FUNCTION_BLOCK TcoInsight_v_5_x_x  EXTENDS TcoIo.TcoPnIoComponent 
VAR_IN_OUT
	inoIoData : TcoInsightIO_v_5_x_x;
END_VAR

VAR
	{attribute addProperty Name "<#Config#>"}
    _config : TcoInsightConfig_v_5_x_x;
	{attribute addProperty Name "<#Status#>"}
	_status : TcoInsightStatus_v_5_x_x;	
END_VAR

VAR
	{attribute addProperty Name "<#UserData#>"}
	_userData 	: TcoInsightUser_v_5_x_x;
	{attribute addProperty Name "<#Results#>"}
	_results : TcoInsightResults_v_5_x_x;
END_VAR

VAR
	{attribute 'hide'}
    _taskEnabled : BOOL;
	{attribute addProperty Name "<#Restore#>"}
    _restoreTask : TcoCore.TcoTask(THIS^);
	{attribute addProperty Name "<#Update signal states#>"}
    _updateSignalStatesTask : TcoCore.TcoTask(THIS^);
	{attribute addProperty Name "<#Change job by number#>"}
    _changeJobByNumberTask : TcoInsightChangeJobByNumber_v_5_x_x(THIS^);
	{attribute addProperty Name "<#Change job by name#>"}
    _changeJobByNameTask : TcoInsightChangeJobByName_v_5_x_x(THIS^);
	{attribute addProperty Name "<#Clear inspection results#>"}
    _clearInspectionResultsTask : TcoInsightClearInspectionResults_v_5_x_x(THIS^);
	{attribute addProperty Name "<#Set user data#>"}
    _setUserDataTask : TcoInsightSetUserData_v_5_x_x(THIS^);
	{attribute addProperty Name "<#Clear user data#>"}
    _clearUserDataTask : TcoInsightClearUserData_v_5_x_x(THIS^);
	{attribute addProperty Name "<#Soft event#>"}
    _softEventTask : TcoInsightSoftEvent_v_5_x_x(THIS^);
	{attribute addProperty Name "<#Trigger#>"}
    _triggerTask : TcoInsightTrigger_v_5_x_x(THIS^);
END_VAR
VAR
    {attribute 'hide'} 
	_varInfo : __SYSTEM.VAR_INFO;
    {attribute 'hide'} 
	_sb : TcoCore.StringBuilder;
END_VAR

IF InvalidReference() THEN
    RETURN;
END_IF

SUPER^(inPnIoBoxState := THIS^.inoIoData.PnIoBoxState,inPnIoBoxDiag := THIS^.inoIoData.PnIoBoxDiag);

IF NOT SUPER^.ProfinetReady THEN
	THIS^._status.ActionDescription := '<#Not ready for operation by means of Profinet network!#>';	
END_IF

IF SUPER^.ProfinetReady AND THIS^._status.ActionDescription = '<#Not ready for operation by means of Profinet network!#>' THEN
	THIS^._status.ActionDescription := '<#Ready for operation!#>';	
END_IF

CheckIfOnline();

//*************RESTORE********************
_taskEnabled := TRUE;
_restoreTask.Enabled := _taskEnabled;
IF _restoreTask.Execute() THEN
	Restore();
//	UpdateSignalStates();
END_IF
//****************************************

//*************UPDATE*********************
IF _config.UpdateStatesPermanently THEN
	UpdateSignalStates();
END_IF;

_taskEnabled:=SUPER^.ProfinetReady;
_taskEnabled := _taskEnabled AND NOT _restoreTask.Busy ;
_updateSignalStatesTask.Enabled := _taskEnabled;
IF _updateSignalStatesTask.Execute() THEN
	UpdateSignalStates();
END_IF
//****************************************

//*************CHANGE*JOB*BY*NUMBER*******
_taskEnabled:=SUPER^.ProfinetReady;
_taskEnabled := _taskEnabled AND NOT _updateSignalStatesTask.Busy;
_changeJobByNumberTask.Enabled := _taskEnabled;
_changeJobByNumberTask(inoIoData := THIS^.inoIoData,inoConfig := THIS^._config,inoStatus := THIS^._status);
//****************************************

//*************CHANGE*JOB*BY*NAME*********
_taskEnabled:=SUPER^.ProfinetReady;
_taskEnabled := _taskEnabled AND NOT _changeJobByNumberTask.Busy;
_changeJobByNameTask.Enabled := _taskEnabled;
_changeJobByNameTask(inoIoData := THIS^.inoIoData,inoConfig := THIS^._config,inoStatus := THIS^._status);
//****************************************

//*************CLEAR*DATA*****************
_taskEnabled:=SUPER^.ProfinetReady;
_taskEnabled := _taskEnabled AND NOT _changeJobByNameTask.Busy;
_clearInspectionResultsTask.Enabled := _taskEnabled;
_clearInspectionResultsTask(inoIoData := THIS^.inoIoData,inoConfig := THIS^._config,inoStatus := THIS^._status,inoResults := THIS^._results);
//****************************************

//*************CLEAR USER DATA*****************
_taskEnabled:=SUPER^.ProfinetReady;
_taskEnabled := _taskEnabled AND NOT _setUserDataTask.Busy  ;
_clearUserDataTask.Enabled := _taskEnabled;
_clearUserDataTask(inoIoData := THIS^.inoIoData,inoConfig := THIS^._config,inoStatus := THIS^._status,inoUserData := THIS^._userData);
//****************************************

//*************SET USER DATA*****************
_taskEnabled:=SUPER^.ProfinetReady;
_taskEnabled := _taskEnabled AND NOT _changeJobByNameTask.Busy AND NOT _clearInspectionResultsTask.Busy AND NOT _triggerTask.Busy ;
_setUserDataTask.Enabled := _taskEnabled;
_setUserDataTask(inoIoData := THIS^.inoIoData,inoConfig := THIS^._config,inoStatus := THIS^._status,inoUserData := THIS^._userData);
//****************************************

//*************SOFT*EVENT*****************
_taskEnabled:=SUPER^.ProfinetReady;
_taskEnabled := _taskEnabled AND THIS^.inoIoData.AcquisitionStatus.Online AND NOT _clearInspectionResultsTask.Busy AND NOT _setUserDataTask.Busy;
_softEventTask.Enabled := _taskEnabled;
_softEventTask(inoIoData := THIS^.inoIoData,inoConfig := THIS^._config,inoStatus := THIS^._status);
//****************************************

//*************TRIGGER********************
_taskEnabled:=SUPER^.ProfinetReady;
_taskEnabled := _taskEnabled AND NOT _clearInspectionResultsTask.Busy AND NOT _setUserDataTask.Busy;
_triggerTask.Enabled :=  _taskEnabled;
_triggerTask(inoIoData := THIS^.inoIoData,inoConfig := THIS^._config,inoStatus := THIS^._status,inoResults := THIS^._results);
//****************************************

(*~
	<docu>
		<summary>
			Clears the inspection results. 		
		</summary>			
	</docu>	
~*)
METHOD ClearInspectionResults : TcoCore.ITcoTaskStatus
ClearInspectionResults := THIS^._clearInspectionResultsTask.Invoke();
END_METHOD

(*~
	<docu>
		<summary>
			Gets the `ClearResultDataTask` task that controls clearing of the results data. 		
		</summary>			
	</docu>	
~*)
PROPERTY ClearInspectionResultsTask : TcoCore.ITcoTaskStatus
GET
ClearInspectionResultsTask := THIS^._clearInspectionResultsTask;
END_GET
END_PROPERTY

(*~
	<docu>
		<summary>
			Clears user data. 		
		</summary>			
	</docu>	
~*)
METHOD ClearUserData : TcoCore.ITcoTaskStatus
ClearUserData := THIS^._clearUserDataTask.Invoke();
END_METHOD

(*~
	<docu>
		<summary>
			Gets the `ClearUserDataTask` task that controls clearing of the user data. 		
		</summary>			
	</docu>	
~*)
PROPERTY ClearUserDataTask : TcoCore.ITcoTaskStatus
GET
ClearUserDataTask := THIS^._clearUserDataTask;
END_GET
END_PROPERTY

(*~
	<docu>
		<summary>
			Gets the configuration of the sensor. 					
		</summary>			
	</docu>	
~*)
PROPERTY Config : REFERENCE TO TcoInsightConfig_v_5_x_x
GET
Config REF= _config;
END_GET
END_PROPERTY

METHOD FB_init : BOOL
VAR_INPUT
	bInitRetains : BOOL; // if TRUE, the retain variables are initialized (warm start / cold start)
	bInCopyCode : BOOL;  // if TRUE, the instance afterwards gets moved into the copy code (online change)
	ParentObject : ITcoObject;
END_VAR
END_METHOD

METHOD GetResultAsByte : BYTE
VAR_INPUT
    inPosition : UINT;
END_VAR
VAR
	_size : UINT;
END_VAR
_size := SIZEOF(GetResultAsByte);

IF (inPosition +_size) > THIS^._config.ResultDataSize THEN
	Messenger.Warning('<#Index of the ResultData in the method GetResultAsByte exceeds the size hardware structure mapped!#>');
	RETURN;
END_IF

IF (inPosition +_size) > TcoVisionParams.MAX_BYTE_ARRAY THEN
	Messenger.Programming('<#Index of the ResultData in the method GetResultAsByte exceeds the defined size!#>');
	RETURN;
END_IF

GetResultAsByte := THIS^._results.InspectionResults[inPosition];
END_METHOD

METHOD GetResultAsDint : DINT
VAR_INPUT
    inPosition : UINT;
END_VAR
VAR
	_index : UINT;
	_size : UINT;
END_VAR
_size := SIZEOF(GetResultAsDint);

IF (inPosition +_size) > THIS^._config.ResultDataSize THEN
	Messenger.Warning('<#Index of the ResultData in the method GetResultAsDint exceeds the size hardware structure mapped!#>');
	RETURN;
END_IF

IF (inPosition +_size) > TcoVisionParams.MAX_BYTE_ARRAY THEN
	Messenger.Programming('<#Index of the ResultData in the method GetResultAsDint exceeds the defined size!#>');
	RETURN;
END_IF

GetResultAsDint := TcoUtilities.TcoBytesToDint(THIS^._config.DataFormat,	THIS^._results.InspectionResults[inPosition],
															THIS^._results.InspectionResults[inPosition+1],
															THIS^._results.InspectionResults[inPosition+2],
															THIS^._results.InspectionResults[inPosition+3]);
END_METHOD

METHOD GetResultAsReal : REAL
VAR_INPUT
    inPosition : UINT;
END_VAR
VAR
	_index : UINT;
	_size : UINT;
END_VAR
_size := SIZEOF(GetResultAsReal);

IF (inPosition +_size) > THIS^._config.ResultDataSize THEN
	Messenger.Warning('<#Index of the ResultData in the method GetResultAsReal exceeds the size hardware structure mapped!#>');
	RETURN;
END_IF

IF (inPosition +_size) > TcoVisionParams.MAX_BYTE_ARRAY THEN
	Messenger.Programming('<#Index of the ResultData in the method GetResultAsReal exceeds the defined size!#>');
	RETURN;
END_IF

GetResultAsReal := TcoUtilities.TcoBytesToReal(THIS^._config.DataFormat,	THIS^._results.InspectionResults[inPosition],
															THIS^._results.InspectionResults[inPosition+1],
															THIS^._results.InspectionResults[inPosition+2],
															THIS^._results.InspectionResults[inPosition+3]);
END_METHOD

METHOD GetResultAsString : STRING
VAR_INPUT
    inPosition : UINT;
	inLength : UINT;
END_VAR
VAR
	_index : UINT;
	_bufferSize : UINT; 
	_resultString : STRING;
END_VAR

IF (inPosition +inLength) > THIS^._config.ResultDataSize THEN
	Messenger.Warning('<#Index of the ResultData in the method GetResultAsString exceeds the size hardware structure mapped!#>');
	RETURN;
END_IF

IF (inPosition +inLength) > TcoVisionParams.MAX_BYTE_ARRAY THEN
	Messenger.Programming('<#Index of the ResultData in the method GetResultAsString exceeds the defined size!#>');
	RETURN;
END_IF

_resultString:='';

IF (inLength>0) THEN 
	FOR	_index := 0 TO inLength-1 BY 1 DO	
		IF(THIS^._results.InspectionResults[inPosition + _index] <> 0) THEN
			_resultString := CONCAT(_resultString, F_ToCHR(THIS^._results.InspectionResults[inPosition + _index]));
		ELSE
			EXIT;	
		END_IF		
	END_FOR;
END_IF

GetResultAsString := _resultString;
END_METHOD

(*~
	<docu>
		<summary>
			Changes the job by its name. 		
		</summary>			
	</docu>	
~*)
METHOD ChangeJobByName : TcoCore.ITcoTaskStatus
VAR_INPUT
	inJobName : STRING;
END_VAR
ChangeJobByName := THIS^._changeJobByNameTask.InvokeWithParameters(inJobName);
END_METHOD

(*~
	<docu>
		<summary>
			Gets the `ClearResultDataTask` task that controls clearing of the results data. 		
		</summary>			
	</docu>	
~*)
PROPERTY ChangeJobByNameTask : TcoCore.ITcoTaskStatus
GET
ChangeJobByNameTask := THIS^._changeJobByNameTask;
END_GET
END_PROPERTY

(*~
	<docu>
		<summary>
			Changes the job by its identification number. 		
		</summary>			
	</docu>	
~*)
METHOD ChangeJobByNumber : TcoCore.ITcoTaskStatus
VAR_INPUT
	inJobNumber : UINT;
END_VAR
ChangeJobByNumber := THIS^._changeJobByNumberTask.InvokeWithParameters(inJobNumber);
END_METHOD

(*~
	<docu>
		<summary>
			Gets the `ClearResultDataTask` task that controls clearing of the results data. 		
		</summary>			
	</docu>	
~*)
PROPERTY ChangeJobByNumberTask : TcoCore.ITcoTaskStatus
GET
ChangeJobByNumberTask := THIS^._changeJobByNumberTask;
END_GET
END_PROPERTY

METHOD INTERNAL CheckIfOnline
VAR_INST
	_onlineTimer : TON;
END_VAR

IF NOT THIS^.inoIoData.AcquisitionStatus.Online THEN
	THIS^._status.CurrentJobName := '';
	THIS^._status.CurrentJobNumber := -1;
END_IF

_onlineTimer(IN:=NOT THIS^.inoIoData.AcquisitionControl.SetOffline AND NOT THIS^.inoIoData.AcquisitionStatus.Online,PT:=T#3S);

Messenger.OnCondition(inoIoData.AcquisitionStatus.OfflineReason0 AND _onlineTimer.Q).Info('<#Camera offline:The vision system$'s job is being modified.#>');
Messenger.OnCondition(inoIoData.AcquisitionStatus.OfflineReason0 AND _onlineTimer.Q).Info('<#Camera offline:A discrete signal is holding the vision system Offline.#>');
Messenger.OnCondition(inoIoData.AcquisitionStatus.OfflineReason0 AND _onlineTimer.Q).Info('<#Camera offline:A communications protocol is holding the vision system Offline.#>');
END_METHOD

METHOD INTERNAL InvalidReference : BOOL
InvalidReference := FALSE;
IF NOT __ISVALIDREF(inoIoData) THEN
	_varInfo :=__VARINFO(inoIoData);
	Messenger.Programming(_sb.Clear().Append('<#Invalid reference: #>').Append(_varInfo.Symbol).ToString());
    InvalidReference := TRUE;
END_IF
END_METHOD

PROPERTY LastResultData : TcoInsightResults_v_5_x_x
GET
LastResultData := THIS^._results;
END_GET
END_PROPERTY

(*~
	<docu>
		<summary>
			Restores this instance to the Ready state. Can be called explicitly or from within one of the restore mechanisms.	
		</summary>			
	</docu>	
~*)
METHOD Restore : ITcoRestorable
_updateSignalStatesTask.Restore();
_changeJobByNumberTask.Restore();
_changeJobByNameTask.Restore();
_clearInspectionResultsTask.Restore();
_softEventTask.Restore();
_triggerTask.Restore();
_clearUserDataTask.Restore();
_setUserDataTask.Restore();

Tc2_System.MEMSET(destAddr:= ADR(THIS^._results.InspectionResults) , fillByte:= 0 , n:= SIZEOF(THIS^._results.InspectionResults));
Tc2_System.MEMSET(destAddr:= ADR(THIS^._userData.UserData) , fillByte:= 0 , n:= SIZEOF(THIS^._userData.UserData));


THIS^._results.InspectionId := 0;
THIS^._results.ResultCode := 0;
	
IF InvalidReference() THEN
    RETURN;
END_IF

Tc2_System.MEMSET(destAddr:= ADR(THIS^.inoIoData) , fillByte:= 0 , n:= SIZEOF(THIS^.inoIoData));

_status.ActionDescription := '<#Restore executed!#>';
_restoreTask.Restore();
END_METHOD

(*~
	<docu>
		<summary>
		    Custom service (manual, maintenance) logic.
			This method must be implemented in derived class.
		</summary>			
	</docu>	
~*)
METHOD PROTECTED ServiceMode
END_METHOD

(*~
	<docu>
		<summary>
			Set user data. 		
		</summary>			
	</docu>	
~*)
METHOD SetUserData : TcoCore.ITcoTaskStatus
SetUserData := THIS^._setUserDataTask.Invoke();
END_METHOD

METHOD SetUserDataAsByte : BOOL;
VAR_INPUT
	inValue : BYTE;
	inPosition : UINT;	
END_VAR
VAR
	_bufferSize : UINT; 
	_size : UINT; 
END_VAR
SetUserDataAsByte := FALSE;

_size := SIZEOF(inValue);

_bufferSize := SIZEOF(THIS^._userData.UserData)/SIZEOF(THIS^._userData.UserData[0]);

IF (inPosition +_size) > THIS^._config.UserDataSize THEN
	Messenger.Info('<#Index of UserData in method SetUserDataAsByte exceeds the size hardware structure mapped#>');
	RETURN;
END_IF

IF (inPosition +_size) > _bufferSize THEN
	Messenger.Info('<#Index of UserData in method SetUserDataAsByte exceeds the defined size#>');
	RETURN;
END_IF

THIS^._userData.UserData[inPosition]:=inValue;

SetUserDataAsByte := TRUE;
END_METHOD

METHOD SetUserDataAsDint : BOOL
VAR_INPUT
	inValue : DINT;
	inPosition : UINT;	
END_VAR
VAR
	_index : UINT;
	_size : UINT;
	_bufferSize : UINT; 
END_VAR
SetUserDataAsDint := FALSE;

_size := SIZEOF(inValue);

_bufferSize := SIZEOF(THIS^._userData.UserData)/SIZEOF(THIS^._userData.UserData[0]);

IF (inPosition +_size) > THIS^._config.UserDataSize THEN
	Messenger.Info('<#Index of UserData in method SetUserDataAsDint exceeds the size hardware structure mapped#>');
	RETURN;
END_IF

IF (inPosition +_size) > _bufferSize THEN
	Messenger.Info('<#Index of UserData in method SetUserDataAsDint exceeds the defined size#>');
	RETURN;
END_IF

TcoDintToBytes(THIS^._config.DataFormat,
				inValue,
				_userData.UserData[inPosition],
				_userData.UserData[inPosition+1],
				_userData.UserData[inPosition+2],
				_userData.UserData[inPosition+3]);	

SetUserDataAsDint := TRUE;
END_METHOD

METHOD SetUserDataAsReal : BOOL
VAR_INPUT
	inValue : DINT;
	inPosition : UINT;	
END_VAR
VAR
	_index : UINT;
	_size : UINT;
	_bufferSize : UINT; 
END_VAR
SetUserDataAsReal := FALSE;

_size := SIZEOF(inValue);

_bufferSize := SIZEOF(THIS^._userData.UserData)/SIZEOF(THIS^._userData.UserData[0]);

IF (inPosition +_size) > THIS^._config.UserDataSize THEN
	Messenger.Info('<#Index of UserData in method SetUserDataAsReal exceeds the size hardware structure mapped#>');
	RETURN;
END_IF

IF (inPosition +_size) > _bufferSize THEN
	Messenger.Info('<#Index of UserData in method SetUserDataAsReal exceeds the defined size#>');
	RETURN;
END_IF

	
TcoRealToBytes(THIS^._config.DataFormat,
				inValue,
				_userData.UserData[inPosition],
				_userData.UserData[inPosition+1],
				_userData.UserData[inPosition+2],
				_userData.UserData[inPosition+3]);			

SetUserDataAsReal := TRUE;
END_METHOD

METHOD SetUserDataAsString : BOOL
VAR_INPUT
	inValue : STRING;
	inPosition : UINT;	
END_VAR
VAR
	_index : UINT;
	_size : UINT;
	_bufferSize : UINT; 
END_VAR
SetUserDataAsString := FALSE;

_size := LEN(inValue);

_bufferSize := SIZEOF(THIS^._userData.UserData)/SIZEOF(THIS^._userData.UserData[0]);

IF (inPosition +_size) > THIS^._config.UserDataSize THEN
	Messenger.Info('<#Index of UserData in method SetUserDataAsString exceeds the size hardware structure mapped#>');
	RETURN;
END_IF

IF (inPosition +_size) > _bufferSize THEN
	Messenger.Info('<#Index of UserData in method SetUserDataAsString exceeds the defined size#>');
	RETURN;
END_IF

FOR	_index := 1 TO _size BY 1 DO	
	_userData.UserData[inPosition + _index-1] := F_ToASC(MID(inValue,1,_index));
END_FOR;

FOR	_index := inPosition +_size TO _bufferSize BY 1 DO	
	_userData.UserData[_index] := 0;
END_FOR;

SetUserDataAsString := TRUE;
END_METHOD

(*~
	<docu>
		<summary>
			Gets the `SetUserDataTask` task that controls to set of the user data. 		
		</summary>			
	</docu>	
~*)
PROPERTY SetUserDataTask : TcoCore.ITcoTaskStatus
GET
SetUserDataTask := THIS^._setUserDataTask;
END_GET
END_PROPERTY

(*~
	<docu>
		<summary>
			Executes the soft event. 		
		</summary>			
	</docu>	
~*)
METHOD SoftEvent : TcoCore.ITcoTaskStatus
VAR_INPUT
    inSoftEventNumber : UINT;
END_VAR
SoftEvent := THIS^._softEventTask.InvokeWithParameters(inSoftEventNumber);
END_METHOD

(*~
	<docu>
		<summary>
			Gets the `ClearResultDataTask` task that controls clearing of the results data. 		
		</summary>			
	</docu>	
~*)
PROPERTY SoftEventTask : TcoCore.ITcoTaskStatus
GET
SoftEventTask := THIS^._softEventTask;
END_GET
END_PROPERTY

(*~
	<docu>
		<summary>
			Gets the status of the sensor. 					
		</summary>			
	</docu>	
~*)
PROPERTY Status : REFERENCE TO TcoInsightStatus_v_5_x_x
GET
Status REF= _status;
END_GET
END_PROPERTY

(*~
	<docu>
		<summary>
			Triggers the reading sequence and waits for results. 		
		</summary>			
	</docu>	
~*)
METHOD Trigger : TcoCore.ITcoTaskStatus
Trigger := THIS^._triggerTask.Invoke();
END_METHOD

(*~
	<docu>
		<summary>
			Gets the `TriggerTask` result. 		
		</summary>			
	</docu>	
~*)
PROPERTY TriggerTask : TcoCore.ITcoTaskStatus
GET
TriggerTask := THIS^._triggerTask;
END_GET
END_PROPERTY

METHOD INTERNAL UpdateSignalStates
_status.SignalStatus.AcquisitionTriggerEnable := inoIoData.AcquisitionControl.AcquisitionTriggerEnable;
_status.SignalStatus.AcquisitionTrigger := inoIoData.AcquisitionControl.AcquisitionTrigger;
_status.SignalStatus.ClearExposureComplete := inoIoData.AcquisitionControl.ClearExposureComplete;
_status.SignalStatus.SetOffline := inoIoData.AcquisitionControl.SetOffline;
  
_status.SignalStatus.EnableResultsBuffering := inoIoData.InspectionControl.EnableResultsBuffering;
_status.SignalStatus.AcknowledgeInspectionResults := inoIoData.InspectionControl.AcknowledgeInspectionResults;
_status.SignalStatus.ExtendedUserDataSet := inoIoData.InspectionControl.ExtendedUserDataSet;
_status.SignalStatus.ExecuteCommand := inoIoData.InspectionControl.ExecuteCommand;
_status.SignalStatus.ClearError := inoIoData.InspectionControl.ClearError;
  
_status.SignalStatus.Command := inoIoData.CommandControl.Command;
  
_status.SignalStatus.TriggerSoftEvent.0 := inoIoData.SoftEventControl.TriggerSoftEvent[0];
_status.SignalStatus.TriggerSoftEvent.1 := inoIoData.SoftEventControl.TriggerSoftEvent[1];
_status.SignalStatus.TriggerSoftEvent.2 := inoIoData.SoftEventControl.TriggerSoftEvent[2];
_status.SignalStatus.TriggerSoftEvent.3 := inoIoData.SoftEventControl.TriggerSoftEvent[3];
_status.SignalStatus.TriggerSoftEvent.4 := inoIoData.SoftEventControl.TriggerSoftEvent[4];
_status.SignalStatus.TriggerSoftEvent.5 := inoIoData.SoftEventControl.TriggerSoftEvent[5];
_status.SignalStatus.TriggerSoftEvent.6 := inoIoData.SoftEventControl.TriggerSoftEvent[6];
_status.SignalStatus.TriggerSoftEvent.7 := inoIoData.SoftEventControl.TriggerSoftEvent[7];
	
_status.SignalStatus.AcquisitionTriggerReady := inoIoData.AcquisitionStatus.AcquisitionTriggerReady;
_status.SignalStatus.AcquisitionTriggerAcknowledge := inoIoData.AcquisitionStatus.AcquisitionTriggerAcknowledge;
_status.SignalStatus.ExposureComplete := inoIoData.AcquisitionStatus.ExposureComplete;
_status.SignalStatus.MissedAcquisition := inoIoData.AcquisitionStatus.MissedAcquisition;
_status.SignalStatus.OfflineReason0 := inoIoData.AcquisitionStatus.OfflineReason0;
_status.SignalStatus.OfflineReason1 := inoIoData.AcquisitionStatus.OfflineReason1;
_status.SignalStatus.OfflineReason2 := inoIoData.AcquisitionStatus.OfflineReason2;
_status.SignalStatus.Online := inoIoData.AcquisitionStatus.Online;
_status.SignalStatus.AcquisitionID := inoIoData.AcquisitionStatus.AcquisitionID;

_status.SignalStatus.SystemBusy := inoIoData.InspectionStatus.SystemBusy;
_status.SignalStatus.InspectionCompleted := inoIoData.InspectionStatus.InspectionCompleted;
_status.SignalStatus.ResultsBufferOverrun := inoIoData.InspectionStatus.ResultsBufferOverrun;
_status.SignalStatus.ResultsValid := inoIoData.InspectionStatus.ResultsValid;
_status.SignalStatus.CommandExecuting := inoIoData.InspectionStatus.CommandExecuting;
_status.SignalStatus.CommandComplete := inoIoData.InspectionStatus.CommandComplete;
_status.SignalStatus.CommandFailed := inoIoData.InspectionStatus.CommandFailed;
_status.SignalStatus.ExtendedUserDataSetAcknowledge := inoIoData.InspectionStatus.ExtendedUserDataSetAcknowledge;
_status.SignalStatus.OverallJobPassFail := inoIoData.InspectionStatus.OverallJobPassFail;
_status.SignalStatus.TestRunReady := inoIoData.InspectionStatus.TestRunReady;
_status.SignalStatus.Error := inoIoData.InspectionStatus.Error;
_status.SignalStatus.ErrorCode := inoIoData.InspectionStatus.ErrorCode;

_status.SignalStatus.CurrentJobID := inoIoData.CommandControl.CurrentJobID;

_status.SignalStatus.TriggerSoftEventAcknowledge.0 := inoIoData.SoftEventControl.TriggerSoftEventAcknowledge[0];
_status.SignalStatus.TriggerSoftEventAcknowledge.1 := inoIoData.SoftEventControl.TriggerSoftEventAcknowledge[1];
_status.SignalStatus.TriggerSoftEventAcknowledge.2 := inoIoData.SoftEventControl.TriggerSoftEventAcknowledge[2];
_status.SignalStatus.TriggerSoftEventAcknowledge.3 := inoIoData.SoftEventControl.TriggerSoftEventAcknowledge[3];
_status.SignalStatus.TriggerSoftEventAcknowledge.4 := inoIoData.SoftEventControl.TriggerSoftEventAcknowledge[4];
_status.SignalStatus.TriggerSoftEventAcknowledge.5 := inoIoData.SoftEventControl.TriggerSoftEventAcknowledge[5];
_status.SignalStatus.TriggerSoftEventAcknowledge.6 := inoIoData.SoftEventControl.TriggerSoftEventAcknowledge[6];
_status.SignalStatus.TriggerSoftEventAcknowledge.7 := inoIoData.SoftEventControl.TriggerSoftEventAcknowledge[7];

_status.SignalStatus.InspectionID := inoIoData.ResultsData.InspectionID;
_status.SignalStatus.ResultCode := inoIoData.ResultsData.ResultCode;

_updateSignalStatesTask.DoneWhen(TRUE);
END_METHOD

PROPERTY UserData : TcoInsightUser_v_5_x_x
GET
UserData := _userData;
END_GET
END_PROPERTY

END_FUNCTION_BLOCK

(* stored: Version 1.1.0.1, ProductVersion 3.1.4024.12
   POU TcoInsight_v_5_x_x: Id {b36dba41-65c9-09aa-02f5-2313aa683dc2}, SpecialFunc None
   Folder _Internals: Id {40d88ad7-ae03-017a-05d9-24612da337bd}
   Folder Operations: Id {42d0a882-7f24-08da-0a00-f03e4d44f85a}
   Folder ResultData: Id {69c0ea1e-0a5f-07ac-2dcf-807d8f23b820}
   Folder States: Id {ca86b13d-4f28-08bb-0f47-84f8e9caefcd}
   Folder Tasks: Id {d3f1ba0f-6a94-07ad-145d-fad2bd01ca0e}
   Folder UserData: Id {b6e57ac1-4435-0688-3216-e8d4a6b9f495}
   Method ClearInspectionResults: Id {ef8962fa-a233-06f4-2210-2d8af175709b}
   Property ClearInspectionResultsTask: Id {8d8fefa6-d752-0e9d-1912-a80b169ef233}
   Get Get: Id {b6a15179-5df8-0d6e-1b51-9398d2fab31f}
   Method ClearUserData: Id {625c0802-8152-0aaa-2ea4-fee184996999}
   Property ClearUserDataTask: Id {578af25a-08a8-0522-31aa-cb2c0964dc0e}
   Get Get: Id {0b1ced55-994c-0ffa-2e64-3ee4f2828c50}
   Property Config: Id {e32f8d76-1a74-0ccc-224c-e9db5cc9a576}
   Get Get: Id {bce6d752-0b26-0b87-125a-730e72a5ca0a}
   Method FB_init: Id {7f208510-b603-07c3-1e51-bbaba95144ef}
   Method GetResultAsByte: Id {229b012a-e07c-09f7-37c9-7e0d54611231}
   Method GetResultAsDint: Id {f78631ce-0b28-029b-3c79-8b570c72f8a5}
   Method GetResultAsReal: Id {15a0d8c5-4660-03a2-2372-1c7ffae688a0}
   Method GetResultAsString: Id {8cbebd56-4f64-0806-093c-54a12437e2d0}
   Method ChangeJobByName: Id {d060e258-4711-083f-2e5f-fd7e215506ca}
   Property ChangeJobByNameTask: Id {9f9bd787-b3c6-05f0-2f81-da95f621af15}
   Get Get: Id {1067b79a-5a4c-0495-2e42-78a896e7d58d}
   Method ChangeJobByNumber: Id {93c62f60-5ccb-093f-1bf1-9b0ec816c0ed}
   Property ChangeJobByNumberTask: Id {10ea4fd1-ba22-0bf8-0a0f-9b0dafc6afe3}
   Get Get: Id {e3790ba3-54b4-0e6d-1342-654760e5a841}
   Method CheckIfOnline: Id {a259a5fe-26bc-40e7-aa53-de1642ff749d}
   Method InvalidReference: Id {c3162119-b996-06e9-2dc7-59f699e9222b}
   Property LastResultData: Id {97762124-4158-0613-21b6-9ba767b94252}
   Get Get: Id {b8b70cbf-6263-0ee7-1d8a-2b09a8021b61}
   Method Restore: Id {0ccd225e-828f-092e-1e14-301fcec7cb64}
   Method ServiceMode: Id {86fa990e-35a2-0992-2a0a-efdfc7c08da5}
   Method SetUserData: Id {5457dc01-fac4-0b42-1737-185529b1def4}
   Method SetUserDataAsByte: Id {3d3891bf-ea7c-4417-babb-4a17a2cd4b2b}
   Method SetUserDataAsDint: Id {8b7643dc-577a-024d-13cd-944d2fee8a30}
   Method SetUserDataAsReal: Id {f4a449e7-c1e7-0a9e-2af7-422d29d39a75}
   Method SetUserDataAsString: Id {5b4200a4-e33d-46ae-aa39-d0a56b524634}
   Property SetUserDataTask: Id {3cfd469d-d30d-0371-2a8f-60bd2e63d711}
   Get Get: Id {376fe7dd-f9b6-07cd-1832-fe63a71e6134}
   Method SoftEvent: Id {966e5f34-d655-0ae7-3c79-57b0e6604da9}
   Property SoftEventTask: Id {14cab0ba-afb8-0a94-1a81-178ea319f9ad}
   Get Get: Id {a98dc00b-68af-0c0c-2e77-958266703660}
   Property Status: Id {884b301f-462d-0b5a-10c0-0bf08336b995}
   Get Get: Id {e080a753-d26d-0878-0500-b6766e154e0e}
   Method Trigger: Id {5aa0db3b-4c5c-0bcd-399c-78ad4bf25313}
   Property TriggerTask: Id {c23205d5-f861-0184-337c-b5fad1b92a5c}
   Get Get: Id {39487498-3f32-05ce-081e-fb2f86d91f86}
   Method UpdateSignalStates: Id {d361a48a-d4a6-0613-237a-4fd373b2cff6}
   Property UserData: Id {0985c5c2-81bd-4346-b100-c946b233a182}
   Get Get: Id {b5e2251f-b3e0-473f-a4e2-67fc8acba436} *)
